TYPE ST_Fahrauftrag :
STRUCT
	Startstockwerk : INT;
	Zielstockwerk : INT;
	istAktiv : BOOL;
	Auftragsnummer : DINT;
END_STRUCT
END_TYPE

(* stored: Version 1.1.0.1
   DUT ST_Fahrauftrag: Id {c46397b2-1b7a-4311-8bd6-25537000d30e} *)
